// TIA Portal V20 export
DATA_BLOCK "GLOBAL_G120D_RBD_HMI_IF_DB"   // DB204
{ S7_Optimized_Access := 'TRUE' }
// stored: AutoNumber false, MemoryReserve 100
   VAR RETAIN
      RBD { S7_SetPoint := 'True'} : Array[0..10] of "H_HMI";
   END_VAR
   VAR
      RBD_G120D { S7_SetPoint := 'True'} : Array[0..6] of "H_Roller2W2S-G120PN";
   END_VAR
BEGIN
   // RBD[1] : ST010RBD01
   // RBD[2] : ST020RBD01
   // RBD[5] : ST030RBD01
   // RBD[6] : ST035RBD01
   // RBD_G120D[1] : ST010RBD01
   // RBD_G120D[2] : ST020RBD01
   // RBD_G120D[5] : ST030RBD01
   // RBD_G120D[6] : ST035RBD01
END_DATA_BLOCK
